FUNCTION_BLOCK EL1722
VAR
	_io : EL1xx2_Data;
	{attribute addProperty Name "WcState"}
	_wcState : WcStateInputToggle;
	{attribute addProperty Name "Info data"}
	_infoData : InfoDataBase;
END_VAR

PROPERTY IO : REFERENCE TO EL1xx2_Data
GET
IO REF= _io;
END_GET
END_PROPERTY

PROPERTY WcState : REFERENCE TO WcStateInputToggle
GET
WcState REF= _wcState;
END_GET
END_PROPERTY

END_FUNCTION_BLOCK

(* stored: Version 1.1.0.1, ProductVersion 3.1.4024.9
   POU EL1722: Id {1319fabe-5d73-0343-23dd-f928a9653c9d}, SpecialFunc None
   Property IO: Id {db88fe8e-5e49-046c-1e19-5fe6aed4444c}
   Get Get: Id {2f660e25-ce00-0845-1b53-7820ec849f0c}
   Property WcState: Id {c7e14249-a9d4-0b71-07cc-9ad63be083aa}
   Get Get: Id {b7f78619-46a4-030e-264c-bc790e950ffd} *)
